INTERFACE ITF_Component_TE2 EXTENDS ITF_BaseComponent

METHOD testMethod : BOOL
VAR_INPUT
END_VAR
END_METHOD

END_INTERFACE

(* stored: Version 1.1.0.1, ProductVersion 3.1.4024.15
   Itf ITF_Component_TE2: Id {6a5f5c57-3e0b-4158-ac5d-4fcc698eda06}
   Method testMethod: Id {b60cdb0e-fe8a-497d-bb9c-c547870b8163} *)
